PROGRAM MAIN
VAR
	// Bedienparameter
	
	// Rezeptparamter
	
	// Grundfunktionen
	Entleeren		:GF_Entleeren;
	Halten			:GF_Halten;
	Pumpen			:GF_Pumpen;
	Zirkulieren		:GF_Zirkulieren;
	Ruehren 		:GF_Ruehren;
	Warten			:GF_Warten;	
	Befuellen		:GF_Befuellen;
	
	// Control- / Statusword
	CW		:RezeptControlWord;
	SW		:RezeptStatusWord;
	
	// Sonstiges
	Leitung			:FB_Leitungswahl;
	
	// Test-Variablen
	Test_Leitung	:INT := 1;
END_VAR

END_PROGRAM

(* stored: Version 1.1.0.1, ProductVersion 3.1.4024.12
   POU MAIN: Id {de090dfa-1e55-4b06-8517-c95a5f22bef4}, SpecialFunc None *)
